INTERFACE PUBLIC CompletedCommands EXTENDS RunningStateCommands, ResettableStateCommands

END_INTERFACE

(* stored: Version 1.1.0.1, ProductVersion 3.1.4026.18
   Itf CompletedCommands: Id {ec0323ba-8561-0e01-188f-98bb79bd5ab9} *)
